// TwinCAT 3 PLC project test_lv1_Communication_opcua
// ProgramVersion: 3.1.4020.1
// libraries:
//   Tc2_Standard, * (Beckhoff Automation GmbH)
//   Tc2_System, * (Beckhoff Automation GmbH)
//   Tc3_Module, * (Beckhoff Automation GmbH)
//   tclib_ph_lv1_comm_opcua, * (Poh)
// project tree:
//   / PlcTask.TcTTO
//   POUs/ MAIN.TcPOU
// (motion and I/O tree: see PLC project ph_lv0)
// real-time tasks:
//   TASK PlcTask: cycle T#10ms, priority 20, ADS port 350

CONFIGURATION test_lv1_Communication_opcua
    RESOURCE PLC ON TwinCAT3
        TASK PlcTask(INTERVAL := T#10ms, PRIORITY := 20);
        PROGRAM MAIN WITH PlcTask : MAIN;
    END_RESOURCE
END_CONFIGURATION

// ---- POUs/MAIN.TcPOU
PROGRAM MAIN
VAR
	c_server : C_OPC_DATASERVER;
	c_client : C_OPC_DATACLIENT(ENCRYPTED_CONNECTION:= FALSE, ENCRYPTION_128_BITS:= FALSE, SERVER_URL:= 'opc.tcp://localhost:4840');
END_VAR

;

END_PROGRAM
